PROGRAM MAIN
VAR
END_VAR

END_PROGRAM

(* stored: Version 1.1.0.1
   POU MAIN: Id {8ef4e1ba-f0be-4cae-8a2d-4d584f3c1237} *)
